FUNCTION_BLOCK CM_SEW_WithBrake EXTENDS CM_Base //IMPLEMENTS I_Motor_base
VAR_INPUT
	i_stSettings : ST_SettingsSEW_WithBrake;
END_VAR
VAR
	// Inputs
	I_bStaReadyForOperation AT %I* : BOOL; // Drive is ready operation (no error)
	
	// Outputs
	Q_bCmdStart AT %Q* : BOOL; // Command to start (+ reset one shot)
	Q_bCmdReverseDirection AT %Q* : BOOL; // Command to reverse direction
	Q_bCmdReleaseBrake AT %Q* : BOOL; // Command to release brake
	Q_nSetTargetSpeed AT %Q* : INT; // Target speed
		
	// Requests
	s_bReqStop : BOOL;
	s_bReqStartForward : BOOL;
	s_bReqStartBackward : BOOL;
	s_bReqReleaseBrake : BOOL;
	s_bReqApplyBrake : BOOL;
	s_bReqReset : BOOL;
	
	// States
	s_bStaReadyForOperation: BOOL;
	s_bStaDriveError: BOOL;
	s_bStaBrakeReleased : BOOL;
	s_bStaMotorStopped : BOOL;
	
	// Setpoints
	s_rTargetSpeed : LREAL; // Target speed [mm/s]
	
	// Timers
	s_tofResetPulse : TOF;
	s_tonMotorStoppedDelay : TON;
	s_tonBrakeReleasedDelay : TON;
	
	// Alarms
	s_fbAlarmHandlerDriveError : FB_AlarmHandler;
	s_fbAlarmHandlerApplyingBrakeNotAllowed : FB_AlarmHandler;
	s_fbAlarmHandlerStartMotorNotAllowed : FB_AlarmHandler;
	
	s_errDriveError : BOOL;
	s_wrnApplyingBrakeNotAllowed : BOOL;
	s_wrnStartMotorNotAllowed : BOOL;
	
	//Hmi
	s_fbHmiBtnManualReleaseBrake: FB_HmiBtn;
	s_fbHmiBtnManualApplyBrake	: FB_HmiBtn;
	s_fbHmiBtnManualForward		: FB_HmiBtn;
	s_fbHmiBtnManualBackward	: FB_HmiBtn;
	s_fbHmiBtnManualStop		: FB_HmiBtn;
	s_fbHmiBtnManualReset		: FB_HmiBtn;
	
	s_fbHmiLedBrakeReleased		: FB_HmiLed;
	s_fbHmiLedMotorStopped		: FB_HmiLed;
	s_fbHmiLedDriveError		: FB_HmiLed;
	
END_VAR

VAR CONSTANT
	cMAX_INT_VALUE : INT := 32767;
END_VAR


SUPER^();

METHOD PROTECTED _m_Alarms : BOOL

IF NOT SUPER^._m_Alarms() THEN
	RETURN;
END_IF

// Set error bits
s_errDriveError := i_bReqEnable AND s_bStaDriveError AND NOT(i_bCmdReset);

// Alarm Handlers
s_fbAlarmHandlerDriveError(
	i_bStaActive := s_errDriveError,
	i_eAlarmLevel := E_AlarmLevel.Alarm,
	i_sAlarmText := CONCAT(i_sCmName, ': Drive - has error (check SEW-drive).'));
	
s_fbAlarmHandlerApplyingBrakeNotAllowed(
	i_bStaActive := s_wrnApplyingBrakeNotAllowed,
	i_eAlarmLevel := E_AlarmLevel.Warning,
	i_sAlarmText := CONCAT(i_sCmName, ': Brake - not allowed to be applied (motor not stopped).'));
	
s_wrnApplyingBrakeNotAllowed R= s_bStaMotorStopped;
	
s_fbAlarmHandlerStartMotorNotAllowed(
	i_bStaActive := s_wrnStartMotorNotAllowed,
	i_eAlarmLevel := E_AlarmLevel.Warning,
	i_sAlarmText := CONCAT(i_sCmName, ': Motor - not allowed to start (brake not released).'));
	
s_wrnStartMotorNotAllowed R= s_bStaBrakeReleased;
	
// Alarm collector	
s_bStaError := 
	s_fbAlarmHandlerDriveError.q_bStaActive;

_m_Alarms := TRUE;
END_METHOD

METHOD PROTECTED _m_Devices : BOOL

IF NOT SUPER^._m_Devices() THEN
	RETURN;
END_IF

//--// Reset request
//--IF s_bStaDoorIsOpened THEN
//--	s_bReqOpen := FALSE;
//--ELSIF s_bStaDoorIsClosed THEN
//--	s_bReqClose := FALSE;	
//--ELSIF s_bStaError THEN
//--	s_bReqOpen := FALSE;
//--	s_bReqClose := FALSE;
//--END_IF

_m_Devices := TRUE;
END_METHOD

METHOD PROTECTED _m_Hmi : BOOL

IF NOT SUPER^._m_Hmi() THEN
	RETURN;
END_IF

//Buttons
s_fbHmiBtnManualReleaseBrake();
s_fbHmiBtnManualApplyBrake();
s_fbHmiBtnManualForward();
s_fbHmiBtnManualBackward();
s_fbHmiBtnManualStop();
s_fbHmiBtnManualReset();

//Led
s_fbHmiLedBrakeReleased(i_bStaLed := s_bStaBrakeReleased);
s_fbHmiLedMotorStopped(i_bStaLed := s_bStaMotorStopped);
s_fbHmiLedDriveError(i_bStaLed := s_bStaDriveError);


{warning '#TODO: Add manual control from hmi'}
		//Is het de bedoeling om op deze plekken de hmi knoppen aan te sturen, OF moet dat gedaan worden in METHOD hmi?		
		s_fbHmiBtnManualApplyBrake.p_bStaVisible := TRUE;
		s_fbHmiBtnManualApplyBrake.p_bStaEnabled := s_bStaMotorStopped;
	
		s_fbHmiBtnManualReleaseBrake.p_bStaVisible := TRUE;
		s_fbHmiBtnManualReleaseBrake.p_bStaEnabled := s_bStaMotorStopped;
		
		s_fbHmiBtnManualStop.p_bStaVisible := TRUE;
		s_fbHmiBtnManualStop.p_bStaEnabled := TRUE;
	
		s_fbHmiBtnManualForward.p_bStaVisible := TRUE;
		s_fbHmiBtnManualForward.p_bStaEnabled := s_bStaMotorStopped;
	
		s_fbHmiBtnManualBackward.p_bStaVisible := TRUE;
		s_fbHmiBtnManualBackward.p_bStaEnabled := s_bStaMotorStopped;
		
		IF s_fbHmiBtnManualApplyBrake.p_osrBtnPress THEN
			m_ReleaseBrake(i_bValue := FALSE);
		END_IF
		
		IF s_fbHmiBtnManualReleaseBrake.p_osrBtnPress THEN
			m_ReleaseBrake(i_bValue := TRUE);
		END_IF
	
		IF s_fbHmiBtnManualReset.p_osrBtnPress THEN
			m_Reset();
		END_IF
			
		IF s_fbHmiBtnManualStop.p_osrBtnPress THEN
			m_Stop();	
		ELSIF s_fbHmiBtnManualForward.p_osrBtnPress THEN
			m_StartForward(i_rTargetSpeed := s_rTargetSpeed);
		ELSIF s_fbHmiBtnManualBackward.p_osrBtnPress THEN
			m_StartBackward(i_rTargetSpeed := s_rTargetSpeed);
		END_IF

_m_Hmi := TRUE;
END_METHOD

METHOD PROTECTED _m_Init : BOOL

IF NOT SUPER^._m_Init() THEN
	RETURN;
END_IF

{warning '#TODO: Not sure if this control module needs initialzation'}
//--s_DOValve.i_stSettings.bCfgDelay 		:= FALSE;
//--s_DOValve.i_stSettings.tmOutputDelay 	:= T#0S;

//Hmi 
	s_fbHmiBtnManualReleaseBrake.p_eButtontype := E_HmiButtonType.PUSHBUTTON;
	s_fbHmiBtnManualReleaseBrake.p_bStaVisible := FALSE;
	s_fbHmiBtnManualReleaseBrake.p_bStaEnabled := FALSE;		
	s_fbHmiBtnManualReleaseBrake.p_sBtnText := 'Release Brake';
	
	s_fbHmiBtnManualApplyBrake.p_eButtontype := E_HmiButtonType.PUSHBUTTON;
	s_fbHmiBtnManualApplyBrake.p_bStaVisible := FALSE;
	s_fbHmiBtnManualApplyBrake.p_bStaEnabled := FALSE;		
	s_fbHmiBtnManualApplyBrake.p_sBtnText := 'Apply Brake';
	
	s_fbHmiBtnManualForward.p_eButtontype := E_HmiButtonType.PUSHBUTTON;
	s_fbHmiBtnManualForward.p_bStaVisible := FALSE;
	s_fbHmiBtnManualForward.p_bStaEnabled := FALSE;		
	s_fbHmiBtnManualForward.p_sBtnText := 'Move Forward';
	
	s_fbHmiBtnManualBackward.p_eButtontype := E_HmiButtonType.PUSHBUTTON;
	s_fbHmiBtnManualBackward.p_bStaVisible := FALSE;
	s_fbHmiBtnManualBackward.p_bStaEnabled := FALSE;		
	s_fbHmiBtnManualBackward.p_sBtnText := 'Move Backward';
	
	s_fbHmiBtnManualStop.p_eButtontype := E_HmiButtonType.PUSHBUTTON;
	s_fbHmiBtnManualStop.p_bStaVisible := FALSE;
	s_fbHmiBtnManualStop.p_bStaEnabled := FALSE;		
	s_fbHmiBtnManualStop.p_sBtnText := 'Stop';

	s_fbHmiBtnManualReset.p_eButtontype := E_HmiButtonType.PUSHBUTTON;
	s_fbHmiBtnManualReset.p_bStaVisible := FALSE;
	s_fbHmiBtnManualReset.p_bStaEnabled := FALSE;		
	s_fbHmiBtnManualReset.p_sBtnText := 'Reset';
	
	s_fbHmiLedBrakeReleased.p_bStaVisible := FALSE;
	s_fbHmiLedBrakeReleased.p_sToHmiDescriptionLed := 'Brake Released';
	
	s_fbHmiLedMotorStopped.p_bStaVisible := FALSE;
	s_fbHmiLedMotorStopped.p_sToHmiDescriptionLed := 'Motor Stopped';
	
	s_fbHmiLedDriveError.p_bStaVisible := FALSE;
	s_fbHmiLedDriveError.p_sToHmiDescriptionLed := 'Drive Error';
	
_m_Init := TRUE;
END_METHOD

METHOD PROTECTED _m_Inputs : BOOL

IF NOT SUPER^._m_Inputs() THEN
	RETURN;
END_IF

s_bStaReadyForOperation := I_bStaReadyForOperation;
s_bStaDriveError := NOT(I_bStaReadyForOperation);

_m_Inputs := TRUE;
END_METHOD

METHOD PROTECTED _m_Outputs : BOOL
VAR
	bCmdStart : BOOL;
END_VAR

IF NOT SUPER^._m_Outputs() THEN
	RETURN;
END_IF

// Generate reset pulse for resetting SEW-drive (via IO, one-shot on start)
s_tofResetPulse(
	IN := s_bReqReset AND s_bStaDriveError AND NOT(s_tofResetPulse.Q),
	PT := i_stSettings.tResetPulseDuration);
s_bReqReset := FALSE;

// Generate time delays for starting motor and brake
s_tonMotorStoppedDelay(
	IN := NOT(Q_bCmdStart),
	PT := i_stSettings.tMotorStoppedDelay,
	Q => s_bStaMotorStopped);

s_tonBrakeReleasedDelay(
	IN := Q_bCmdReleaseBrake,
	PT := i_stSettings.tBrakeReleasedDelay,
	Q => s_bStaBrakeReleased); 
	
Q_bCmdReleaseBrake := (i_bReqEnable AND s_bReqReleaseBrake)
						OR (s_bReqStartForward OR s_bReqStartBackward)
						OR NOT(s_bStaMotorStopped); // Make sure the brake can't be applied when drive is not stopped	

bCmdStart := i_bReqEnable AND (s_bReqStartForward OR s_bReqStartBackward);
Q_bCmdStart := s_tofResetPulse.Q OR (bCmdStart AND s_bStaBrakeReleased); // Make sure that drive can't start when brake is not released	
				
Q_bCmdReverseDirection := i_bReqEnable AND s_bReqStartBackward;

// Write (convert) target speed drive (analog output)
IF i_bReqEnable AND (s_bReqStartForward OR s_bReqStartBackward) THEN
	Q_nSetTargetSpeed := LREAL_TO_INT(s_rTargetSpeed / i_stSettings.rMaxTargetSpeed * cMAX_INT_VALUE);
ELSE
	Q_nSetTargetSpeed := 0;	
END_IF	
	
_m_Outputs := TRUE;
END_METHOD

METHOD PUBLIC m_ApplyBrake : BOOL

IF NOT i_bReqEnable THEN 
	RETURN;
END_IF

s_bReqApplyBrake := TRUE;

m_ApplyBrake := TRUE;
END_METHOD

/// Release brake
METHOD PUBLIC m_ReleaseBrake : BOOL
VAR_INPUT
	i_bValue : BOOL; /// FALSE = apply, TRUE = release
END_VAR

IF NOT i_bReqEnable THEN 
	RETURN;
END_IF

IF i_bValue THEN
	s_bReqReleaseBrake := TRUE;
ELSIF NOT(i_bValue) THEN
	IF s_bStaMotorStopped THEN
		s_bReqReleaseBrake := FALSE;
	ELSE
		{warning: #TODO: Generate warning that }
	END_IF	
END_IF

m_ReleaseBrake := TRUE;
END_METHOD

METHOD PUBLIC m_Reset : BOOL

IF NOT i_bReqEnable THEN 
	RETURN;
END_IF

s_bReqStop := FALSE;
s_bReqStartForward := FALSE;
s_bReqStartBackward := FALSE;
//--s_bReqReleaseBrake := FALSE;
s_bReqReset := TRUE;

m_Reset := TRUE;
END_METHOD

METHOD PUBLIC m_StartBackward : BOOL
VAR_INPUT
	i_rTargetSpeed : LREAL; // Target speed [mm/s]
END_VAR

IF NOT i_bReqEnable THEN 
	RETURN;
END_IF

s_bReqStop := FALSE;
s_bReqStartForward := FALSE;
s_bReqStartBackward := TRUE;
s_bReqReleaseBrake := FALSE;
s_bReqReset := FALSE;

IF i_rTargetSpeed < 0 THEN
	s_rTargetSpeed := 0;
ELSIF i_rTargetSpeed > cMAX_INT_VALUE THEN	
	i_rTargetSpeed := cMAX_INT_VALUE;
ELSE 
	s_rTargetSpeed := i_rTargetSpeed;
END_IF
	
m_StartBackward := TRUE;
END_METHOD

METHOD PUBLIC m_StartForward : BOOL
VAR_INPUT
	i_rTargetSpeed : LREAL; // Target speed [mm/s]
END_VAR

IF NOT i_bReqEnable THEN 
	RETURN;
END_IF

s_bReqStop := FALSE;
s_bReqStartForward := TRUE;
s_bReqStartBackward := FALSE;
s_bReqReleaseBrake := FALSE;
s_bReqReset := FALSE;

IF i_rTargetSpeed < 0 THEN
	s_rTargetSpeed := 0;
ELSIF i_rTargetSpeed > cMAX_INT_VALUE THEN	
	i_rTargetSpeed := cMAX_INT_VALUE;
ELSE 
	s_rTargetSpeed := i_rTargetSpeed;
END_IF

m_StartForward := TRUE;
END_METHOD

METHOD PUBLIC m_Stop : BOOL

IF NOT i_bReqEnable THEN 
	RETURN;
END_IF

s_bReqStop := TRUE;
s_bReqStartForward := FALSE;
s_bReqStartBackward := FALSE;
s_bReqReleaseBrake := FALSE;
s_bReqReset := FALSE;

m_Stop := TRUE;
END_METHOD

{attribute 'monitoring':='call'}
PROPERTY PUBLIC p_bStaBrakeReleased : BOOL
GET

p_bStaBrakeReleased := s_bStaBrakeReleased;
END_GET
END_PROPERTY

{attribute 'monitoring':='call'}
PROPERTY PUBLIC p_bStaMotorRunning : BOOL
GET

p_bStaMotorRunning := s_bStaReadyForOperation AND NOT(s_bStaMotorStopped);
END_GET
END_PROPERTY

{attribute 'monitoring':='call'}
PROPERTY PUBLIC p_bStaMotorStopped : BOOL
GET

p_bStaMotorStopped := s_bStaMotorStopped;
END_GET
END_PROPERTY

END_FUNCTION_BLOCK

(* stored: Version 1.1.0.1, ProductVersion 3.1.4024.12
   POU CM_SEW_WithBrake: Id {d8988437-f8ba-4649-8850-7b7474b271b5}, SpecialFunc None
   Folder Methods: Id {fea5fc79-9587-4159-bfcb-2bdf1bcbabe5}
   Folder Properties: Id {90bb6a76-9d90-4e6c-a11c-e7f0ed29a681}
   Method _m_Alarms: Id {4deaa654-c608-48ef-b852-683d2aa00f57}
   Method _m_Devices: Id {7cf2b106-f168-4b96-b992-17948b9589f2}
   Method _m_Hmi: Id {247a12f4-0dca-4cad-aba1-676ebffdadcb}
   Method _m_Init: Id {e95de6ba-8291-48d3-aa10-18b69b93d9d4}
   Method _m_Inputs: Id {3dd66686-d1af-4a23-8b08-c424814fad43}
   Method _m_Outputs: Id {f0e0fd71-b4a5-4c65-b115-0d3a3aae58a1}
   Method m_ApplyBrake: Id {84406420-53a7-4cd1-828e-c4d2ed555d95}
   Method m_ReleaseBrake: Id {710cca1b-1464-4a44-9af2-adc97e3f5673}
   Method m_Reset: Id {7a4bff47-bee3-4de3-b793-bf5b0f24ba84}
   Method m_StartBackward: Id {49196a88-b792-4b99-9376-81b43964f03b}
   Method m_StartForward: Id {551b77ef-9474-4bb1-9b3d-8c47176aa994}
   Method m_Stop: Id {e9ddf609-54b2-4594-bc3c-53ac00446898}
   Property p_bStaBrakeReleased: Id {9fbced02-9547-4710-b53f-47079111072e}
   Get Get: Id {4b22f759-5b10-4a1a-8c0a-aa7be90f3a40}
   Property p_bStaMotorRunning: Id {05cc9b52-a456-4963-9313-489e38d28904}
   Get Get: Id {48de4f54-9de3-4f86-a416-721c15990310}
   Property p_bStaMotorStopped: Id {a6d82e37-5355-4a67-b5f0-d07baedba186}
   Get Get: Id {88de46fd-3b89-42e4-ad0b-d4b96e0ab51a} *)
